// TIA Portal V19 export
TYPE "ItemStatus_UDT"
   STRUCT
      SPARE1 : Bool;
      SPARE2 : Bool;
      SPARE3 : Bool;
      Auto : Bool;
      Process_Mirror : Bool;
      AlarmResetTimer : Byte;
   END_STRUCT;
END_TYPE
